# EPICS substitutions: iocBoot/iocgalil/galil_dmc_ctrl.substitutions
# $File: //ASP/Dev/SBS/4_Controls/4_3_Network_Infrastructure/4_3_1_Comms_Common_Services/sw/device_drivers/Galil/1-5/galilTestApp/Db/galil_ctrl_extras.substitutions $
# $Revision: #2 $
# $DateTime: 2012/03/20 11:55:19 $
# $Author: cliftm $
#
# Description
# Substitution file for readback/commands that are in addition to features provided by motorRecord
#
# This library is free software; you can redistribute it and/or
# modify it under the terms of the GNU Lesser General Public
# Licence as published by the Free Software Foundation; either
# version 2.1 of the Licence, or (at your option) any later version.
#
# This library is distributed in the hope that it will be useful,
# but WITHOUT ANY WARRANTY; without even the implied warranty of
# MERCHANTABILITY or FITNESS FOR A PARTICULAR PURPOSE.  See the GNU
# Lesser General Public Licence for more details.
#
# You should have received a copy of the GNU Lesser General Public
# Licence along with this library; if not, write to the Free Software
# Foundation, Inc., 51 Franklin St, Fifth Floor, Boston, MA 02110-1301 USA.
#
# Contact details:
# mark.clift@synchrotron.org.au
# 800 Blackburn Road, Clayton, Victoria 3168, Australia.
#

# P    - PV prefix
# PORT - Asyn port name
# SCAN - Scan period for monitor records.  Use passive when only epics will change value (default)
#      - Periodic scan will slow controller update performance (poller)
# DEFAULT_LIMITTYPE = 0 Normally open, 1 Normally closed
# DEFAULT_HOMETYPE = 0 Normally open, 1 Normally closed
# PREC - precision

file "$(TOP)/db/galil_dmc_ctrl.template"
{
pattern
{   P,	     PORT,    SCAN, 	  DEFAULT_HOMETYPE, DEFAULT_LIMITTYPE, PREC}
 {  "CEL:GALIL", "Galil", "Passive",  1,                1,                 5 }
}

# end
